% RSLogix 500 project Practise-3.RSS, saved by version 8.30.00.16 %
PROJECT "UNTITLED"    % processor: MicroLogix 1000 %

PROGRAM FILES
  LAD 2 "MAIN_PROG"  7 rungs
  LAD 3 "USER_FAULT"  1 rungs
  LAD 4 "HSC_INT"  1 rungs
  LAD 5 "STI_INT"  1 rungs
  LAD 6, 7, 8, 9, 10, 11, 12, 13, 14, 15, 16: only END

DATA FILES
  O0 OUTPUT  1 elements
  I1 INPUT  2 elements
  S2 STATUS  33 elements
  B3 BINARY  32 elements
  T4 TIMER  40 elements
  C5 COUNTER  32 elements
  R6 CONTROL  16 elements
  N7 INTEGER  105 elements

LADDER 2 "MAIN_PROG"
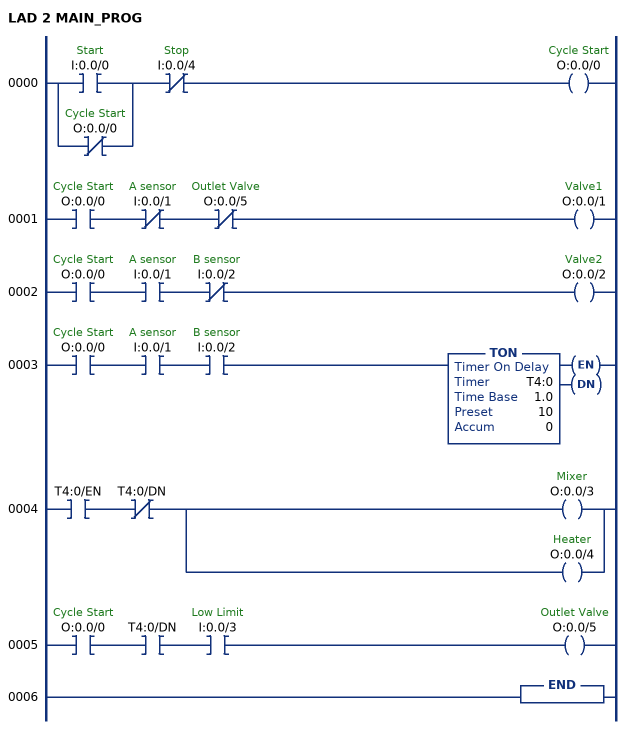
% Rung: 0 %
SOR BST XIC I:0.0/0 NXB XIO O:0.0/0 BND XIO I:0.0/4 OTE O:0.0/0 EOR
%   I:0.0/0  "Start" %
%   O:0.0/0  "Cycle Start" %
%   I:0.0/4  "Stop" %
% Rung: 1 %
SOR XIC O:0.0/0 XIO I:0.0/1 XIO O:0.0/5 OTE O:0.0/1 EOR
%   O:0.0/0  "Cycle Start" %
%   I:0.0/1  "A sensor" %
%   O:0.0/5  "Outlet Valve" %
%   O:0.0/1  "Valve1" %
% Rung: 2 %
SOR XIC O:0.0/0 XIC I:0.0/1 XIO I:0.0/2 OTE O:0.0/2 EOR
%   O:0.0/0  "Cycle Start" %
%   I:0.0/1  "A sensor" %
%   I:0.0/2  "B sensor" %
%   O:0.0/2  "Valve2" %
% Rung: 3 %
SOR XIC O:0.0/0 XIC I:0.0/1 XIC I:0.0/2 TON T4:0 1.0 10 0 EOR
%   O:0.0/0  "Cycle Start" %
%   I:0.0/1  "A sensor" %
%   I:0.0/2  "B sensor" %
% Rung: 4 %
SOR XIC T4:0/EN XIO T4:0/DN BST OTE O:0.0/3 NXB OTE O:0.0/4 BND EOR
%   O:0.0/3  "Mixer" %
%   O:0.0/4  "Heater" %
% Rung: 5 %
SOR XIC O:0.0/0 XIC T4:0/DN XIC I:0.0/3 OTE O:0.0/5 EOR
%   O:0.0/0  "Cycle Start" %
%   I:0.0/3  "Low Limit" %
%   O:0.0/5  "Outlet Valve" %
% Rung: 6 %
SOR END EOR

DATA TABLE (non-zero values as saved)
DATA T4
% .PRE .ACC %
% T4:0 % 10 0
